// TIA Portal V15.1 export
// export: Created 2020-06-12T07:35:54.0224609Z, ExportSetting None, DisplayName Totally Integrated Automation Portal, DisplayVersion V15.1, DisplayName TIA Portal Openness, DisplayVersion V15.1, DisplayName STEP 7 Professional, DisplayVersion V15.1, DisplayName STEP 7 Safety, DisplayVersion V15.1, DisplayName WinCC Advanced, DisplayVersion V15.1
FUNCTION "RCW_Fans" : Void   // FC179, FBD
TITLE = RCW: air cooling fans controller
{ S7_Optimized_Access := 'TRUE' }
// stored: SetENOAutomatically False
   VAR_TEMP
      tFanTimeOff : Time;
   END_VAR
BEGIN

REGION Network 1: Fans are ready
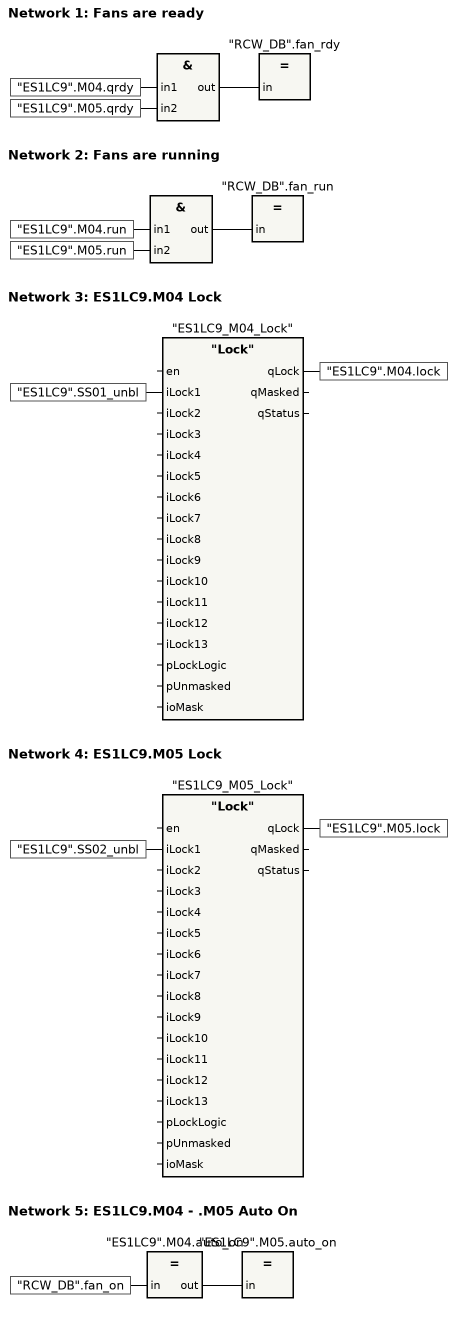
   "RCW_DB".fan_rdy := "ES1LC9".M04.qrdy AND "ES1LC9".M05.qrdy;
END_REGION

REGION Network 2: Fans are running
   "RCW_DB".fan_run := "ES1LC9".M04.run AND "ES1LC9".M05.run;
END_REGION

REGION Network 3: ES1LC9.M04 Lock
   "ES1LC9_M04_Lock"(iLock1 := "ES1LC9".SS01_unbl, qLock => "ES1LC9".M04.lock);   // "Lock"
END_REGION

REGION Network 4: ES1LC9.M05 Lock
   "ES1LC9_M05_Lock"(iLock1 := "ES1LC9".SS02_unbl, qLock => "ES1LC9".M05.lock);   // "Lock"
END_REGION

REGION Network 5: ES1LC9.M04 - .M05 Auto On
   "ES1LC9".M04.auto_on := "RCW_DB".fan_on;
   "ES1LC9".M05.auto_on := "RCW_DB".fan_on;
END_REGION

REGION Network 6: ES1LC9.M04 - .M05 : speed set
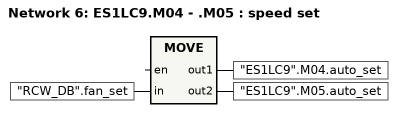
   "ES1LC9".M04.auto_set := "RCW_DB".fan_set;
   "ES1LC9".M05.auto_set := "RCW_DB".fan_set;
END_REGION
END_FUNCTION
